TYPE (* A Structure with 2 BOOLS *)
  (* Version 1.0, 2024-02-21, Franz Höpfinger, HR Agrartechnik GmbH *)
  PACKAGE logiBUS::utils::conversion::types;
  ST02X : STRUCT
    X_00 : BOOL; (* BIT 00 *)
    X_01 : BOOL; (* BIT 01 *)
  END_STRUCT;
END_TYPE
